// TIA Portal V19 export
VAR_GLOBAL   // PLC tag table "Standard_IO"
   I_IPBDoorAccesRequest AT %I100.0 : Bool;   // Illuminate push button acces request   {ExternalAccessible false}
   I_IPBCloseDoor AT %I100.1 : Bool;   // Illuminate push button close door   {ExternalAccessible false}
   I_EStopState AT %I100.2 : Bool;   // Entry door AU state   {ExternalAccessible false}
   I_DoorClosed AT %I100.3 : Bool;   // Entry door state 1   {ExternalAccessible false}
   I_BoltTongueInserted AT %I100.4 : Bool;   // Entry door state 2   {ExternalAccessible false}
   I_GuardLocked AT %I100.5 : Bool;   // Entry door state 3   {ExternalAccessible false}
   I_FaultPresent AT %I100.6 : Bool;   // Entry door state 4   {ExternalAccessible false}
   I_PSAirLeftRobotOk AT %I101.0 : Bool;   // Air supply robot 1 Ok   {ExternalAccessible false}
   I_PSAirRightRobotOk AT %I101.1 : Bool;   // Air supply robot 2 Ok   {ExternalAccessible false}
   I_PSAirSuctionUnitOk AT %I101.2 : Bool;   // Air supply suction unit Ok   {ExternalAccessible false}
   I_FanDriveRunning AT %I101.4 : Bool;   // Suction unit - Fan Drive Running   {ExternalAccessible false}
   I_DustBagFull AT %I101.5 : Bool;   // Suction unit - Dust bag full   {ExternalAccessible false}
   I_FanDriveFault AT %I101.6 : Bool;   // Suction unit - Fan Drive fault   {ExternalAccessible false}
   I_SequencerFault AT %I101.7 : Bool;   // Suction unit - Sequencer in fault   {ExternalAccessible false}
   O_IPBDoorAccesRequest AT %Q100.0 : Bool;   // Illuminate push button acces request   {ExternalAccessible false}
   O_IPBCloseDoor AT %Q100.1 : Bool;   // Illuminate push button close door   {ExternalAccessible false}
   O_ResetDoorFault AT %Q100.2 : Bool;   // Reset fault on door   {ExternalAccessible false}
   O_SignalToweGreenLight AT %Q100.4 : Bool;   // Light towers - green light   {ExternalAccessible false}
   O_SignalToweOrangeLight AT %Q100.5 : Bool;   // Light towers - orange light   {ExternalAccessible false}
   O_SignalToweRedLight AT %Q100.6 : Bool;   // Light towers - red light   {ExternalAccessible false}
   O_SignalToweHorn AT %Q100.7 : Bool;   // Light towers - horn   {ExternalAccessible false}
   O_StartVacuum AT %Q101.4 : Bool;   // Suction unit - Vacuum On   {ExternalAccessible false}
   O_StopVacuum AT %Q101.5 : Bool;   // Suction unit - Vacuum Off   {ExternalAccessible false}
   O_TeepTrackCycleTimeR1 AT %Q102.0 : Bool;   // Alstom Teep track Cycle Time Robot 1 (Left)   {ExternalAccessible false}
   O_TeepTrackStartStopR1 AT %Q102.1 : Bool;   // Alstom Teep track Start and Stop Robot 1 (Left)   {ExternalAccessible false}
   O_LockDoor AT %Q101.0 : Bool;   // Lock acces door   {ExternalAccessible false}
   OST_SendLeft AT %Q106.0 : "stMasterToSlave";   // Send information to left slave PLC   {ExternalAccessible false}
   OST_SendRight AT %Q234.0 : "stMasterToSlave";   // Send information to right slave PLC   {ExternalAccessible false}
   IST_ReceiveLeft AT %I106.0 : "stSlaveToMaster";   // Receive information from left slave PLC   {ExternalAccessible false}
   IST_ReceiveRight AT %I234.0 : "stSlaveToMaster";   // Receive information from right slave PLC   {ExternalAccessible false}
   I_FanFault AT %I102.0 : Bool;   // Suction unit - Fan fault   {ExternalAccessible false}
   I_ValveMotorFault AT %I102.1 : Bool;   // Suction unit - Valve Motor Fault   {ExternalAccessible false}
   IB_100 AT %IB100 : SInt;   //    {ExternalWritable false}
   IB_101 AT %IB101 : SInt;   //    {ExternalWritable false}
   IB_102 AT %IB102 : SInt;   //    {ExternalWritable false}
   IB_103 AT %IB103 : SInt;   //    {ExternalWritable false}
   OB_100 AT %QB100 : SInt;   //    {ExternalWritable false}
   OB_101 AT %QB101 : SInt;   //    {ExternalWritable false}
   OB_102 AT %QB102 : SInt;   //    {ExternalWritable false}
   OB_103 AT %QB103 : SInt;   //    {ExternalWritable false}
   O_TeepTrackCycleTimeR2 AT %Q102.2 : Bool;   // Alstom Teep track Cycle Time Robot 2 (Right)   {ExternalAccessible false}
   O_TeepTrackStartStopR2 AT %Q102.3 : Bool;   // Alstom Teep track Start and Stop Robot 2 (Right)   {ExternalAccessible false}
END_VAR
